(* Logix 5000 project; controller cal1615 1756-L62 rev 20.19; software revision 20.05; part 62 of 81 *)
(* tags used below, declared in another part *)
   FAULT : BOOL;   // Fault AFI
   HMI : BOOL;   // AFI HMI
   p01r09_pb_global_reset : BOOL;   // System Modes PB: Global Fault Reset
   p26_ao_dia_a : REAL;   // Upper Poly Letoff Analog Input Letoff A Diameter
   p26_ao_dia_b : REAL;   // Upper Poly Letoff Analog Input Letoff B Diameter
   p26_dint_to_hmi : DINT[16];   // Upper Poly Letoff Dint to HMI
   p26_ltf_a_sensor_input_max : REAL;
   p26_ltf_a_sensor_input_min : REAL;
   p26_ltf_a_sensor_output_max : REAL;
   p26_ltf_a_sensor_output_min : REAL;
   p26_ltf_b_sensor_input_max : REAL;
   p26_ltf_b_sensor_input_min : REAL;
   p26_ltf_b_sensor_output_max : REAL;
   p26_ltf_b_sensor_output_min : REAL;
   p26_ula_prs_input_max : REAL;
   p26_ula_prs_input_min : REAL;
   p26_ula_prs_output_max : REAL;
   p26_ula_prs_output_min : REAL;
   p26_ulb_prs_input_max : REAL;
   p26_ulb_prs_input_min : REAL;
   p26_ulb_prs_output_max : REAL;
   p26_ulb_prs_output_min : REAL;
   p26r01 : routine;   // Upper Poly Letoff
   p26r02 : routine;   // Upper Poly Letoff
   p26r02_fault_exists : BOOL;
   p26r02_timer_fault : TIMER[4];   // Upper Poly Letoff Misc Control Fault Delay
   p26r02_timer_warning : TIMER[4];   // Upper Poly Letoff Misc Control Warning Delay
   p26r02_unack_fault : BOOL;   // Upper Poly Letoff Misc Control Unacknowledged Fault Exists
   p26r02_unack_warning : BOOL;   // Upper Poly Letoff Misc Control Unacknowledged Warning Exists
   p26r02_warning_exists : BOOL;
   p26r03 : routine;   // Upper Poly Letoff Input
   p26r03_a_radius : REAL;
   p26r03_ai_dia_a_sensor : REAL;
   p26r03_ai_dia_b_sensor : REAL;
   p26r03_b_radius : REAL;
   p26r03_ltf_a_sensor_scp : SYS_SCP;   // Upper Poly Letoff Analog Input Diameter A Sensor Scaling
   p26r03_ltf_b_sensor_scp : SYS_SCP;   // Upper Poly Letoff Analog Input Letoff B Diameter Sensor Scaling
   p26r03_timer_fault : TIMER[4];   // Lower Poly Letoff Input Fault Delay
   p26r03_timer_warning : TIMER[4];   // Lower Poly Letoff Input Warning Delay
   p26r03_upper_A_tension_on : BOOL;
   p26r03_upper_B_tension_on : BOOL;
   p26r03_upper_poly_a_distance : REAL;
   p26r03_upper_poly_b_distance : REAL;
   p26r04 : routine;   // Upper Poly Letoff Output
   p26r04_timer_fault : TIMER[4];   // Lower Poly Letoff Output Fault Delay
   p26r04_timer_warning : TIMER[4];   // Lower Poly Letoff Output Warning Delay
   p26r04_ula_prs_scp : SYS_SCP;   // Upper Poly Lefoff Analog Output Letoff A Brake Pressure
   p26r04_ulb_prs_scp : SYS_SCP;   // Upper Poly Lefoff Analog Output Letoff B Brake Pressure
   p26r05 : routine;   // Upper Poly Letoff Dint to HMI
   p26r05_timer_fault : TIMER[4];   // Lower Poly Letoff Dint to HMI Fault Delay
   p26r06 : routine;   // Upper Poly Letoff Real to HMI
   p26r07 : routine;   // Upper Poly Letoff Alarms
   p26r08 : routine;   // Upper Poly Letoff Warnings
   p26r09 : routine;   // Upper Poly Letoff Modes
   p26r10 : routine;   // Upper Poly Letoff Tension
   p26r10_ula_selected_tension : REAL;   // Upper Poly Letoff Tension A Selected Tension
   p26r10_ulb_selected_tension : REAL;   // Upper Poly Letoff Tension B Selected Tension

PROGRAM P26_Upper_Poly_Letoff   (* main routine R01_Main *)

ROUTINE R01_Main   (* ladder *)
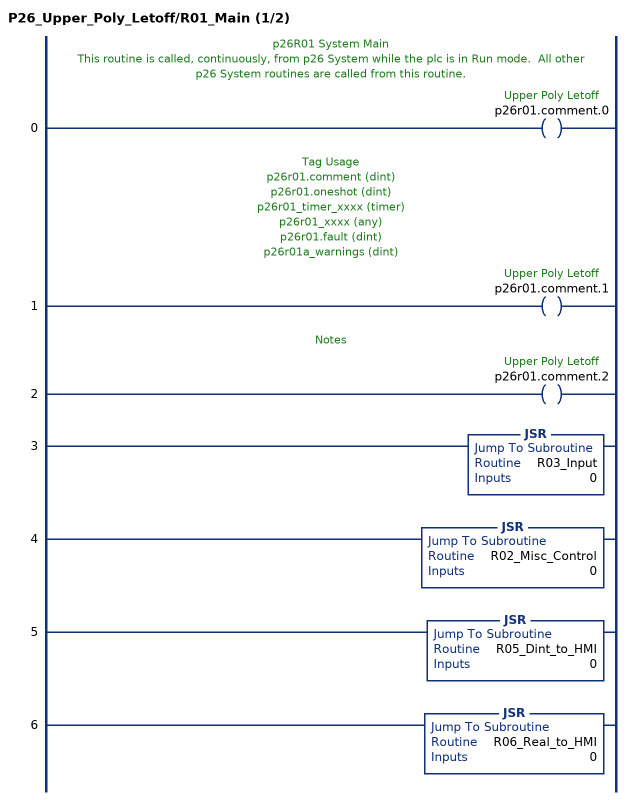
   // p26R01 System Main
   // This routine is called, continuously, from p26 System while the plc is in Run mode.  All other p26 System routines are called from this routine.
   0: OTE(p26r01.comment.0);
   // Tag Usage
   // p26r01.comment (dint)
   // p26r01.oneshot (dint)
   // p26r01_timer_xxxx (timer)
   // p26r01_xxxx (any)
   // p26r01.fault (dint)
   // p26r01a_warnings (dint)
   1: OTE(p26r01.comment.1);
   // Notes
   2: OTE(p26r01.comment.2);
   3: JSR(R03_Input,0);
   4: JSR(R02_Misc_Control,0);
   5: JSR(R05_Dint_to_HMI,0);
   6: JSR(R06_Real_to_HMI,0);
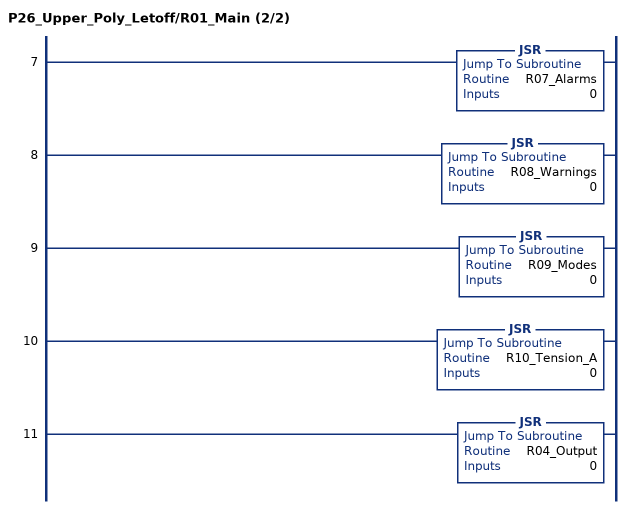
   7: JSR(R07_Alarms,0);
   8: JSR(R08_Warnings,0);
   9: JSR(R09_Modes,0);
   10: JSR(R10_Tension_A,0);
   11: JSR(R04_Output,0);
END_ROUTINE

ROUTINE R02_Misc_Control   (* ladder *)
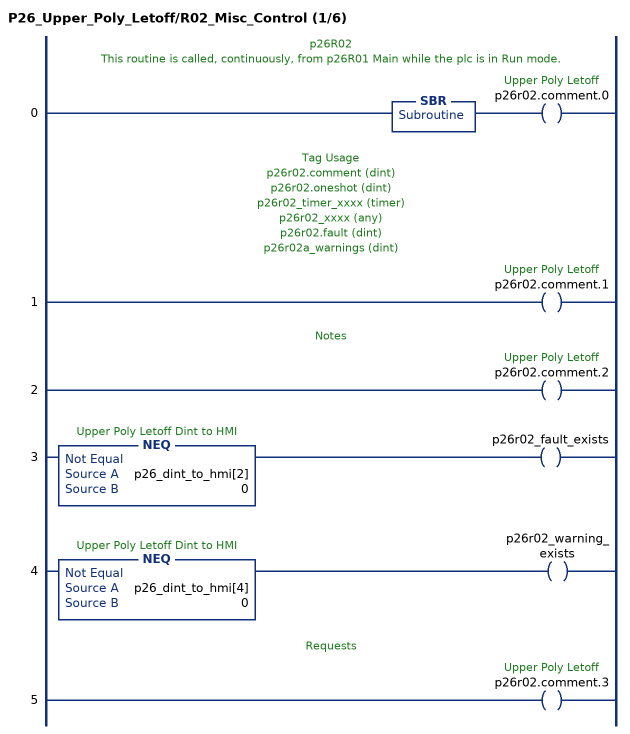
   // p26R02
   // This routine is called, continuously, from p26R01 Main while the plc is in Run mode.
   0: SBR()OTE(p26r02.comment.0);
   // Tag Usage
   // p26r02.comment (dint)
   // p26r02.oneshot (dint)
   // p26r02_timer_xxxx (timer)
   // p26r02_xxxx (any)
   // p26r02.fault (dint)
   // p26r02a_warnings (dint)
   1: OTE(p26r02.comment.1);
   // Notes
   2: OTE(p26r02.comment.2);
   3: NEQ(p26_dint_to_hmi[2],0)OTE(p26r02_fault_exists);
   4: NEQ(p26_dint_to_hmi[4],0)OTE(p26r02_warning_exists);
   // Requests
   5: OTE(p26r02.comment.3);
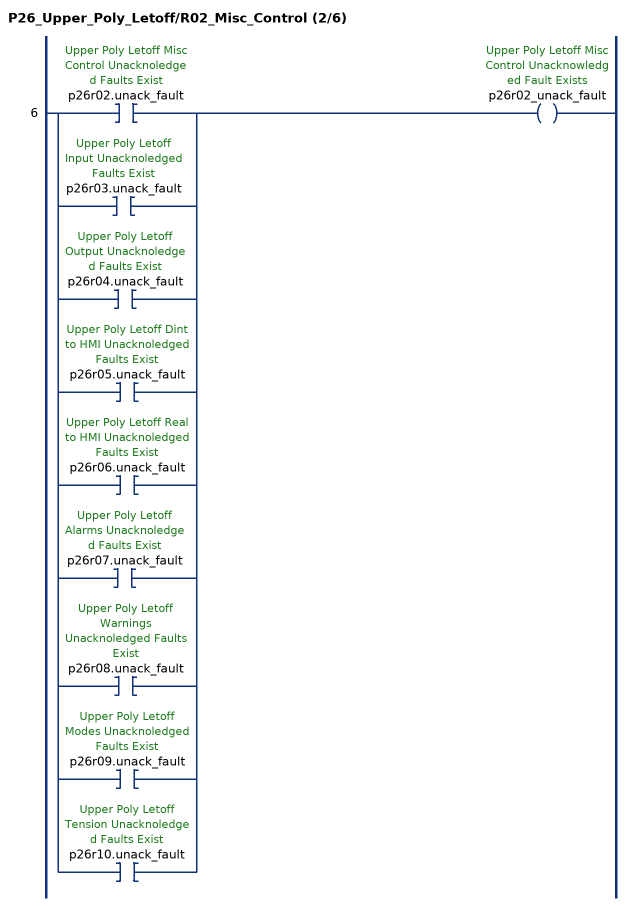
   6: [XIC(p26r02.unack_fault) ,XIC(p26r03.unack_fault) ,XIC(p26r04.unack_fault) ,XIC(p26r05.unack_fault) ,XIC(p26r06.unack_fault) ,XIC(p26r07.unack_fault) ,XIC(p26r08.unack_fault) ,XIC(p26r09.unack_fault) ,XIC(p26r10.unack_fault) ]OTE(p26r02_unack_fault);
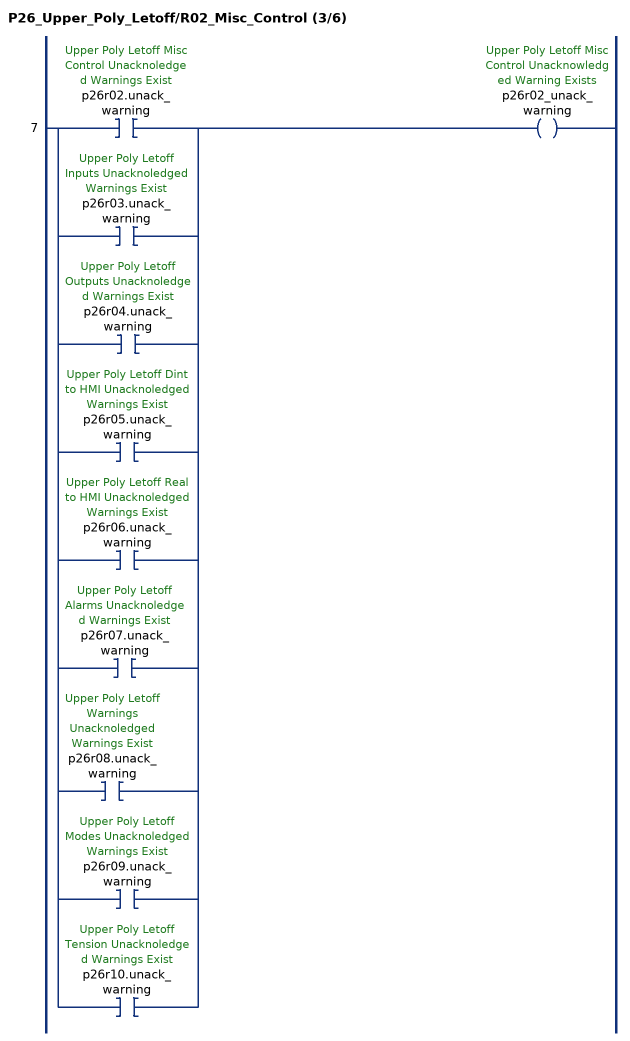
   7: [XIC(p26r02.unack_warning) ,XIC(p26r03.unack_warning) ,XIC(p26r04.unack_warning) ,XIC(p26r05.unack_warning) ,XIC(p26r06.unack_warning) ,XIC(p26r07.unack_warning) ,XIC(p26r08.unack_warning) ,XIC(p26r09.unack_warning) ,XIC(p26r10.unack_warning) ]OTE(p26r02_unack_warning);
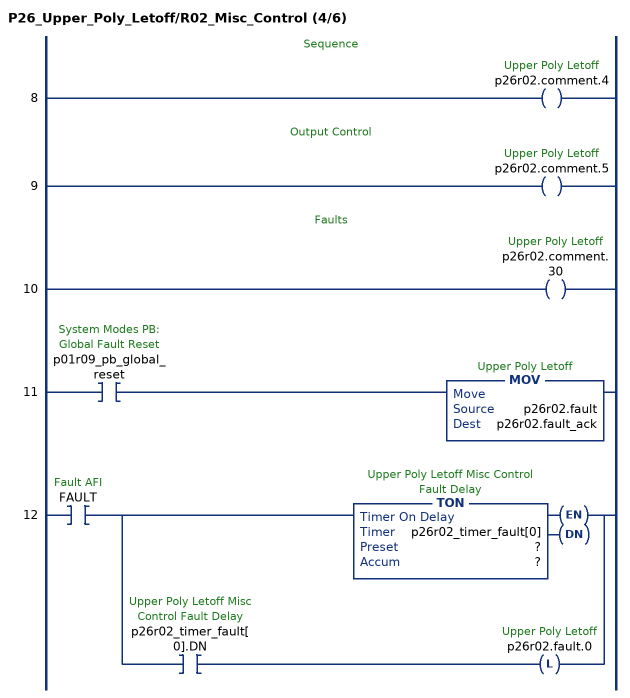
   // Sequence
   8: OTE(p26r02.comment.4);
   // Output Control
   9: OTE(p26r02.comment.5);
   // Faults
   10: OTE(p26r02.comment.30);
   11: XIC(p01r09_pb_global_reset)MOV(p26r02.fault,p26r02.fault_ack);
   12: XIC(FAULT)[TON(p26r02_timer_fault[0],?,?) ,XIC(p26r02_timer_fault[0].DN) OTL(p26r02.fault.0) ];
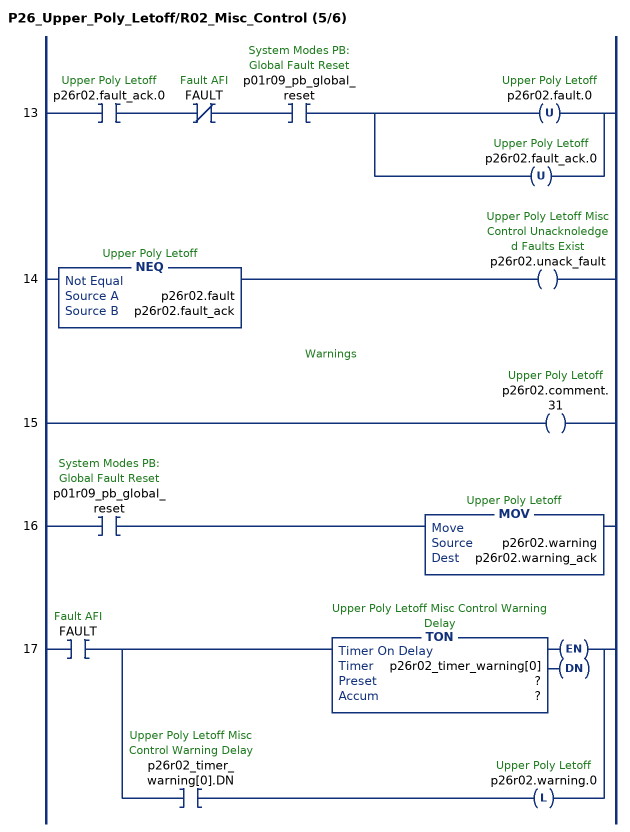
   13: XIC(p26r02.fault_ack.0)XIO(FAULT)XIC(p01r09_pb_global_reset)[OTU(p26r02.fault.0) ,OTU(p26r02.fault_ack.0) ];
   14: NEQ(p26r02.fault,p26r02.fault_ack)OTE(p26r02.unack_fault);
   // Warnings
   15: OTE(p26r02.comment.31);
   16: XIC(p01r09_pb_global_reset)MOV(p26r02.warning,p26r02.warning_ack);
   17: XIC(FAULT)[TON(p26r02_timer_warning[0],?,?) ,XIC(p26r02_timer_warning[0].DN) OTL(p26r02.warning.0) ];
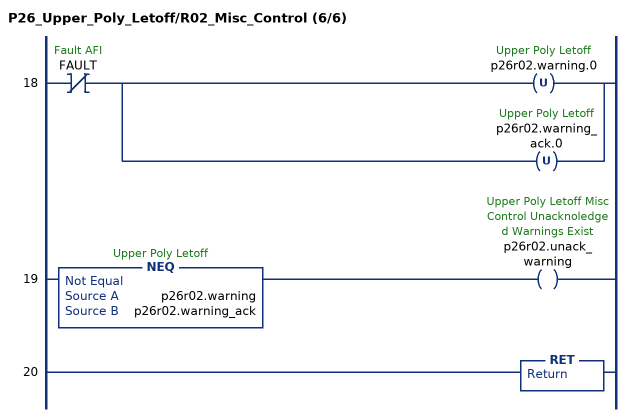
   18: XIO(FAULT)[OTU(p26r02.warning.0) ,OTU(p26r02.warning_ack.0) ];
   19: NEQ(p26r02.warning,p26r02.warning_ack)OTE(p26r02.unack_warning);
   20: RET();
END_ROUTINE

ROUTINE R03_Input   (* ladder *)
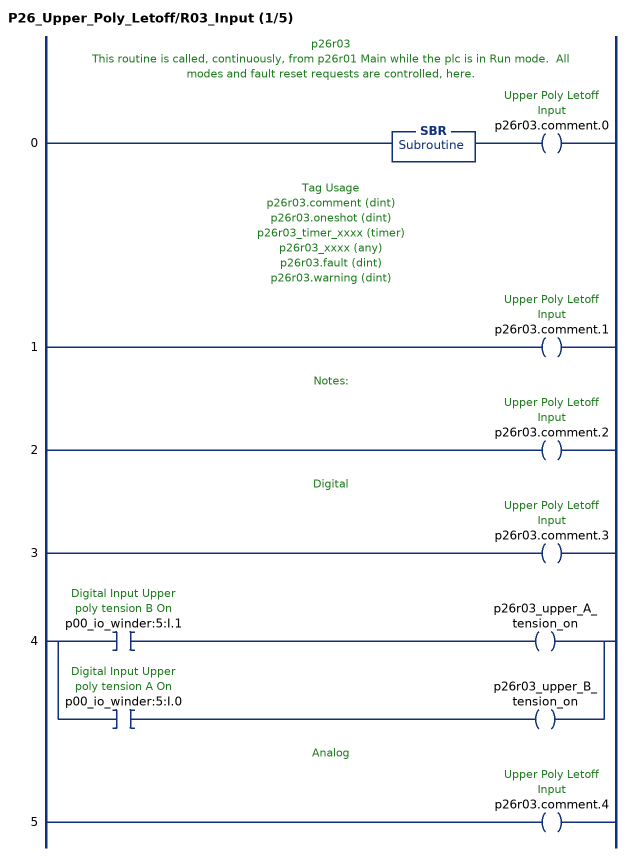
   // p26r03
   // This routine is called, continuously, from p26r01 Main while the plc is in Run mode.  All modes and fault reset requests are controlled, here.
   0: SBR()OTE(p26r03.comment.0);
   // Tag Usage
   // p26r03.comment (dint)
   // p26r03.oneshot (dint)
   // p26r03_timer_xxxx (timer)
   // p26r03_xxxx (any)
   // p26r03.fault (dint)
   // p26r03.warning (dint)
   1: OTE(p26r03.comment.1);
   // Notes:
   2: OTE(p26r03.comment.2);
   // Digital
   3: OTE(p26r03.comment.3);
   4: [XIC(p00_io_winder:5:I.1) OTE(p26r03_upper_A_tension_on) ,XIC(p00_io_winder:5:I.0) OTE(p26r03_upper_B_tension_on) ];
   // Analog
   5: OTE(p26r03.comment.4);
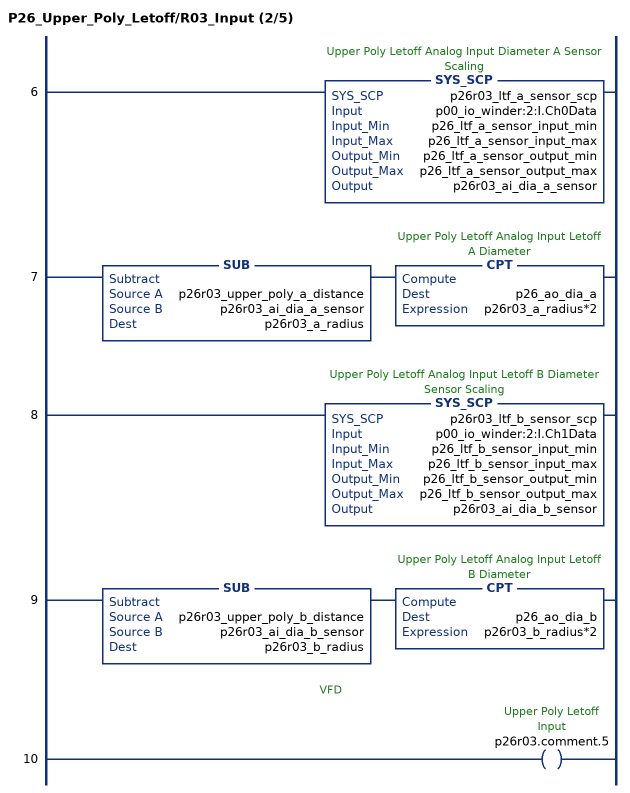
   6: SYS_SCP(p26r03_ltf_a_sensor_scp,p00_io_winder:2:I.Ch0Data,p26_ltf_a_sensor_input_min,p26_ltf_a_sensor_input_max,p26_ltf_a_sensor_output_min,p26_ltf_a_sensor_output_max,p26r03_ai_dia_a_sensor);
   7: SUB(p26r03_upper_poly_a_distance,p26r03_ai_dia_a_sensor,p26r03_a_radius)CPT(p26_ao_dia_a,p26r03_a_radius*2);
   8: SYS_SCP(p26r03_ltf_b_sensor_scp,p00_io_winder:2:I.Ch1Data,p26_ltf_b_sensor_input_min,p26_ltf_b_sensor_input_max,p26_ltf_b_sensor_output_min,p26_ltf_b_sensor_output_max,p26r03_ai_dia_b_sensor);
   9: SUB(p26r03_upper_poly_b_distance,p26r03_ai_dia_b_sensor,p26r03_b_radius)CPT(p26_ao_dia_b,p26r03_b_radius*2);
   // VFD
   10: OTE(p26r03.comment.5);
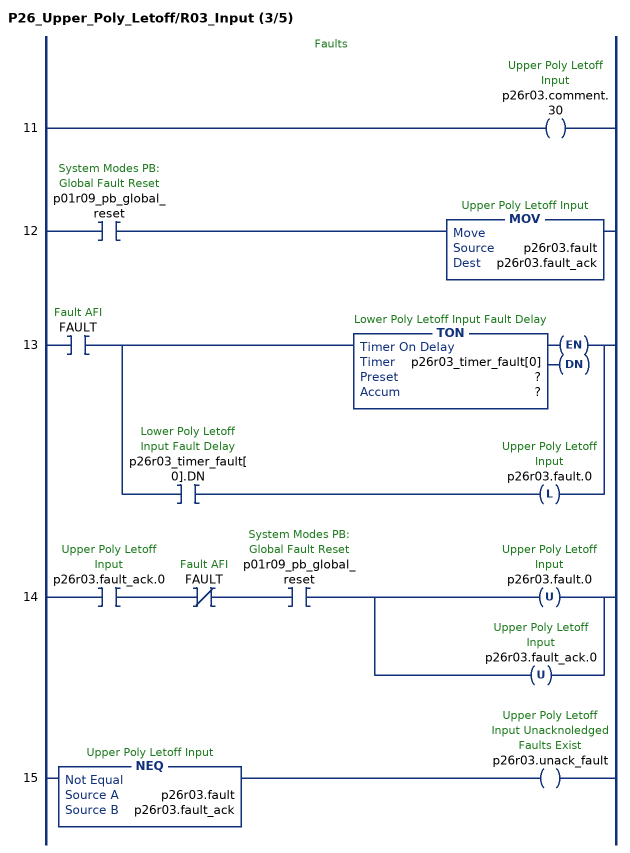
   // Faults
   11: OTE(p26r03.comment.30);
   12: XIC(p01r09_pb_global_reset)MOV(p26r03.fault,p26r03.fault_ack);
   13: XIC(FAULT)[TON(p26r03_timer_fault[0],?,?) ,XIC(p26r03_timer_fault[0].DN) OTL(p26r03.fault.0) ];
   14: XIC(p26r03.fault_ack.0)XIO(FAULT)XIC(p01r09_pb_global_reset)[OTU(p26r03.fault.0) ,OTU(p26r03.fault_ack.0) ];
   15: NEQ(p26r03.fault,p26r03.fault_ack)OTE(p26r03.unack_fault);
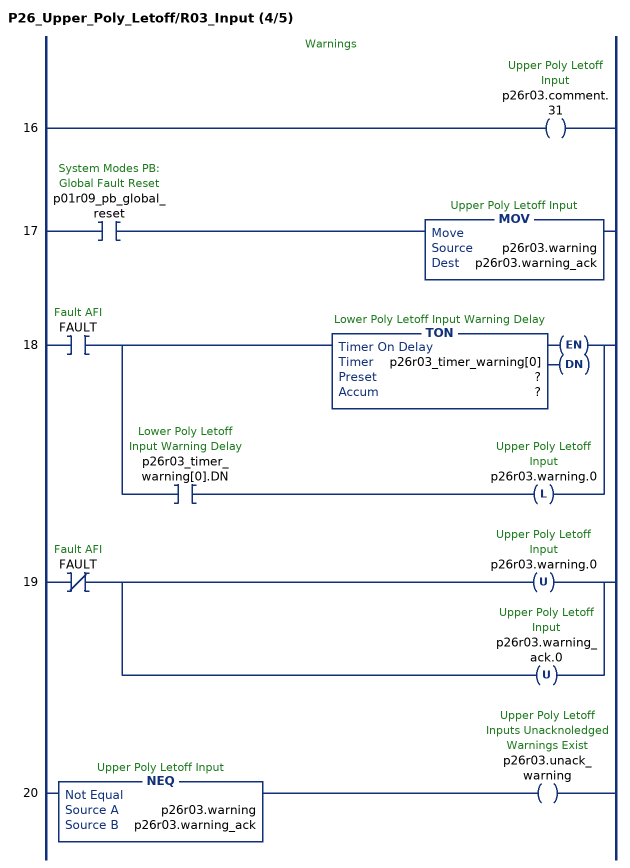
   // Warnings
   16: OTE(p26r03.comment.31);
   17: XIC(p01r09_pb_global_reset)MOV(p26r03.warning,p26r03.warning_ack);
   18: XIC(FAULT)[TON(p26r03_timer_warning[0],?,?) ,XIC(p26r03_timer_warning[0].DN) OTL(p26r03.warning.0) ];
   19: XIO(FAULT)[OTU(p26r03.warning.0) ,OTU(p26r03.warning_ack.0) ];
   20: NEQ(p26r03.warning,p26r03.warning_ack)OTE(p26r03.unack_warning);
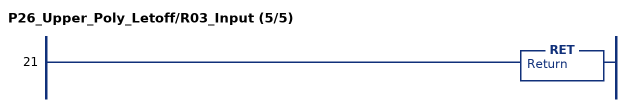
   21: RET();
END_ROUTINE

ROUTINE R04_Output   (* ladder *)
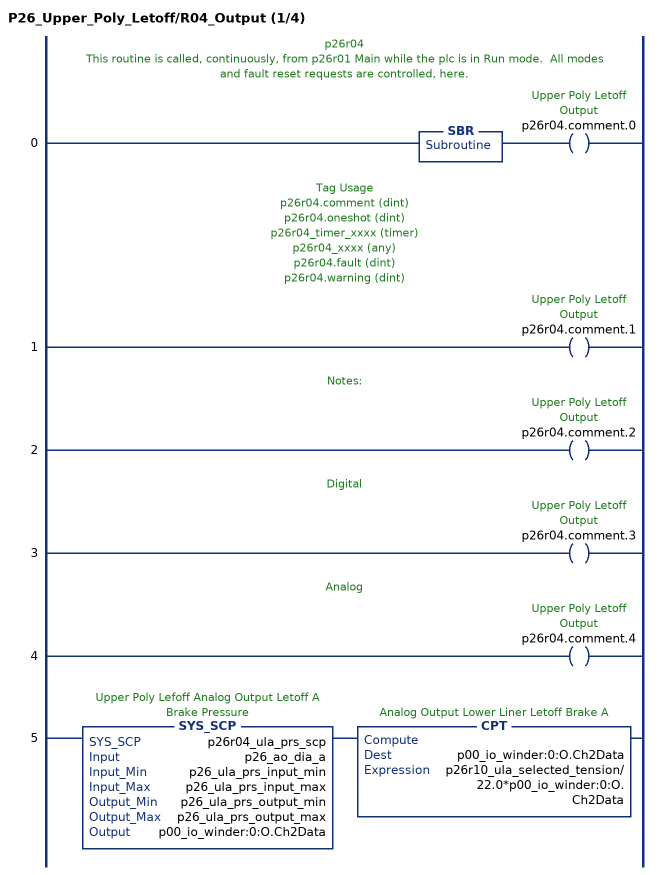
   // p26r04
   // This routine is called, continuously, from p26r01 Main while the plc is in Run mode.  All modes and fault reset requests are controlled, here.
   0: SBR()OTE(p26r04.comment.0);
   // Tag Usage
   // p26r04.comment (dint)
   // p26r04.oneshot (dint)
   // p26r04_timer_xxxx (timer)
   // p26r04_xxxx (any)
   // p26r04.fault (dint)
   // p26r04.warning (dint)
   1: OTE(p26r04.comment.1);
   // Notes:
   2: OTE(p26r04.comment.2);
   // Digital
   3: OTE(p26r04.comment.3);
   // Analog
   4: OTE(p26r04.comment.4);
   5: SYS_SCP(p26r04_ula_prs_scp,p26_ao_dia_a,p26_ula_prs_input_min,p26_ula_prs_input_max,p26_ula_prs_output_min,p26_ula_prs_output_max,p00_io_winder:0:O.Ch2Data)CPT(p00_io_winder:0:O.Ch2Data,p26r10_ula_selected_tension/22.0*p00_io_winder:0:O.Ch2Data);
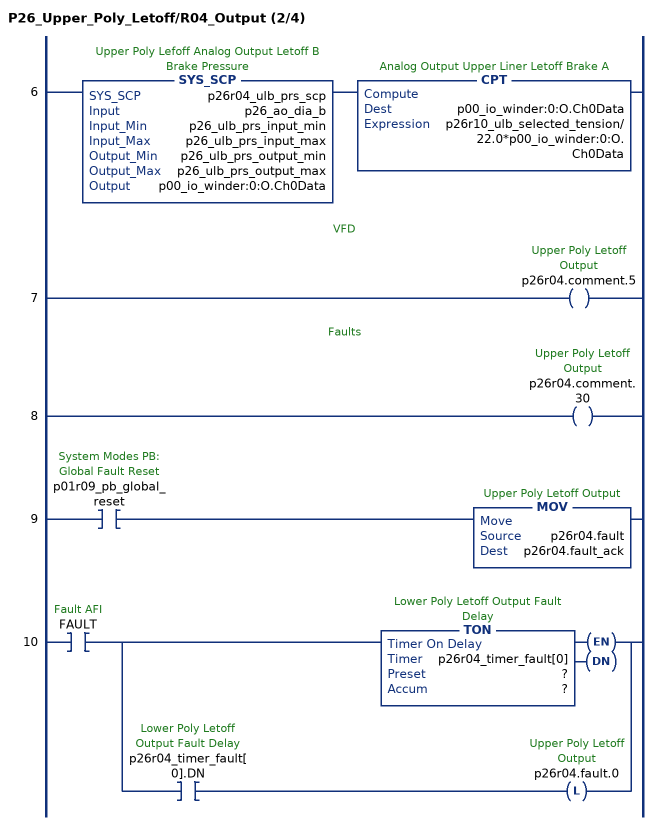
   6: SYS_SCP(p26r04_ulb_prs_scp,p26_ao_dia_b,p26_ulb_prs_input_min,p26_ulb_prs_input_max,p26_ulb_prs_output_min,p26_ulb_prs_output_max,p00_io_winder:0:O.Ch0Data)CPT(p00_io_winder:0:O.Ch0Data,p26r10_ulb_selected_tension/22.0*p00_io_winder:0:O.Ch0Data);
   // VFD
   7: OTE(p26r04.comment.5);
   // Faults
   8: OTE(p26r04.comment.30);
   9: XIC(p01r09_pb_global_reset)MOV(p26r04.fault,p26r04.fault_ack);
   10: XIC(FAULT)[TON(p26r04_timer_fault[0],?,?) ,XIC(p26r04_timer_fault[0].DN) OTL(p26r04.fault.0) ];
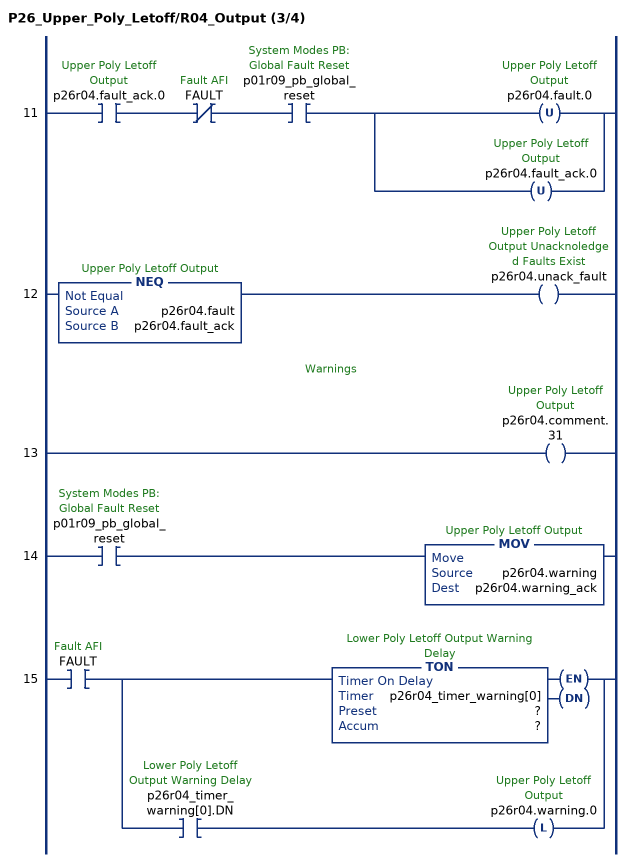
   11: XIC(p26r04.fault_ack.0)XIO(FAULT)XIC(p01r09_pb_global_reset)[OTU(p26r04.fault.0) ,OTU(p26r04.fault_ack.0) ];
   12: NEQ(p26r04.fault,p26r04.fault_ack)OTE(p26r04.unack_fault);
   // Warnings
   13: OTE(p26r04.comment.31);
   14: XIC(p01r09_pb_global_reset)MOV(p26r04.warning,p26r04.warning_ack);
   15: XIC(FAULT)[TON(p26r04_timer_warning[0],?,?) ,XIC(p26r04_timer_warning[0].DN) OTL(p26r04.warning.0) ];
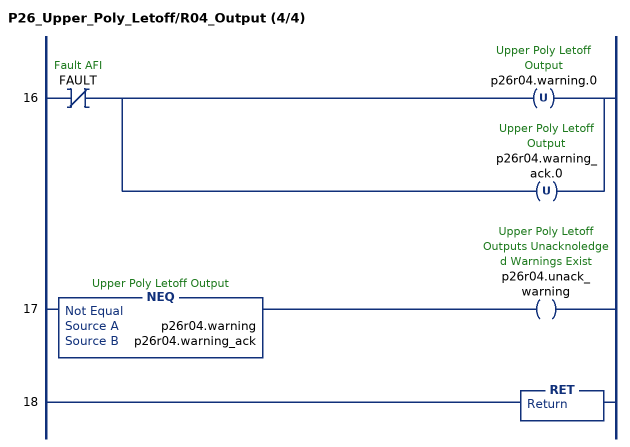
   16: XIO(FAULT)[OTU(p26r04.warning.0) ,OTU(p26r04.warning_ack.0) ];
   17: NEQ(p26r04.warning,p26r04.warning_ack)OTE(p26r04.unack_warning);
   18: RET();
END_ROUTINE

ROUTINE R05_Dint_to_HMI   (* ladder *)
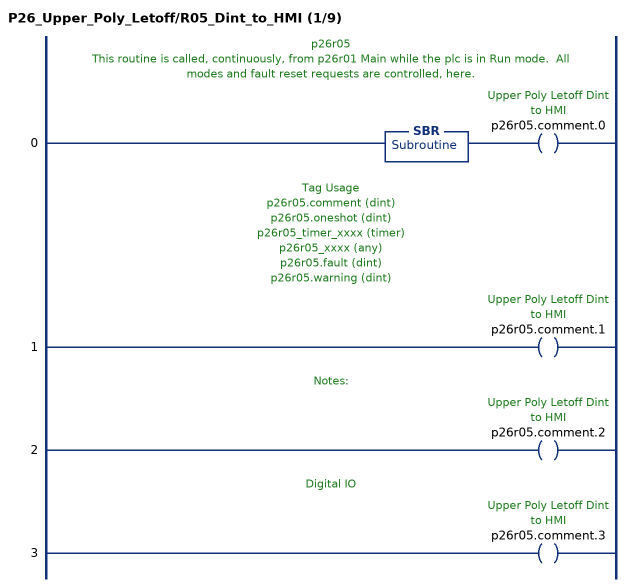
   // p26r05
   // This routine is called, continuously, from p26r01 Main while the plc is in Run mode.  All modes and fault reset requests are controlled, here.
   0: SBR()OTE(p26r05.comment.0);
   // Tag Usage
   // p26r05.comment (dint)
   // p26r05.oneshot (dint)
   // p26r05_timer_xxxx (timer)
   // p26r05_xxxx (any)
   // p26r05.fault (dint)
   // p26r05.warning (dint)
   1: OTE(p26r05.comment.1);
   // Notes:
   2: OTE(p26r05.comment.2);
   // Digital IO
   3: OTE(p26r05.comment.3);
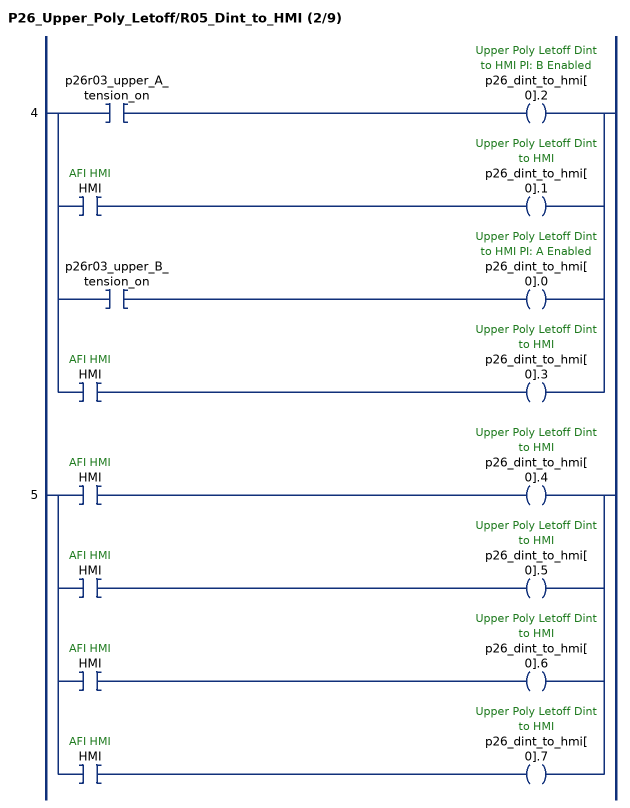
   4: [XIC(p26r03_upper_A_tension_on) OTE(p26_dint_to_hmi[0].2) ,XIC(HMI) OTE(p26_dint_to_hmi[0].1) ,XIC(p26r03_upper_B_tension_on) OTE(p26_dint_to_hmi[0].0) ,XIC(HMI) OTE(p26_dint_to_hmi[0].3) ];
   5: [XIC(HMI) OTE(p26_dint_to_hmi[0].4) ,XIC(HMI) OTE(p26_dint_to_hmi[0].5) ,XIC(HMI) OTE(p26_dint_to_hmi[0].6) ,XIC(HMI) OTE(p26_dint_to_hmi[0].7) ];
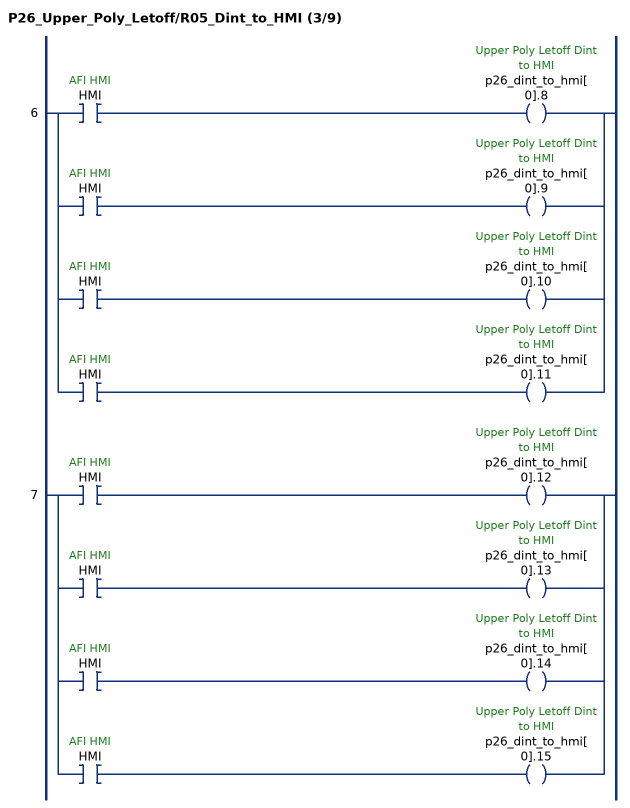
   6: [XIC(HMI) OTE(p26_dint_to_hmi[0].8) ,XIC(HMI) OTE(p26_dint_to_hmi[0].9) ,XIC(HMI) OTE(p26_dint_to_hmi[0].10) ,XIC(HMI) OTE(p26_dint_to_hmi[0].11) ];
   7: [XIC(HMI) OTE(p26_dint_to_hmi[0].12) ,XIC(HMI) OTE(p26_dint_to_hmi[0].13) ,XIC(HMI) OTE(p26_dint_to_hmi[0].14) ,XIC(HMI) OTE(p26_dint_to_hmi[0].15) ];
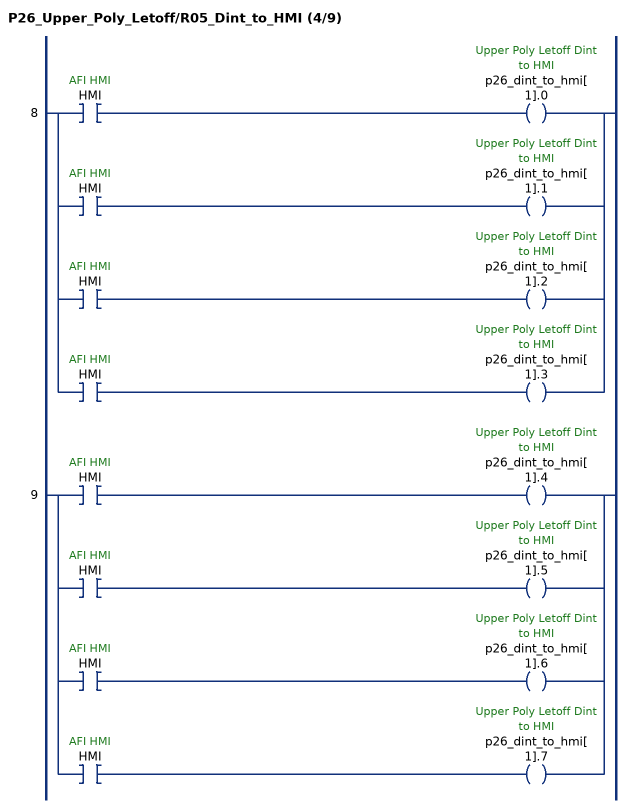
   8: [XIC(HMI) OTE(p26_dint_to_hmi[1].0) ,XIC(HMI) OTE(p26_dint_to_hmi[1].1) ,XIC(HMI) OTE(p26_dint_to_hmi[1].2) ,XIC(HMI) OTE(p26_dint_to_hmi[1].3) ];
   9: [XIC(HMI) OTE(p26_dint_to_hmi[1].4) ,XIC(HMI) OTE(p26_dint_to_hmi[1].5) ,XIC(HMI) OTE(p26_dint_to_hmi[1].6) ,XIC(HMI) OTE(p26_dint_to_hmi[1].7) ];
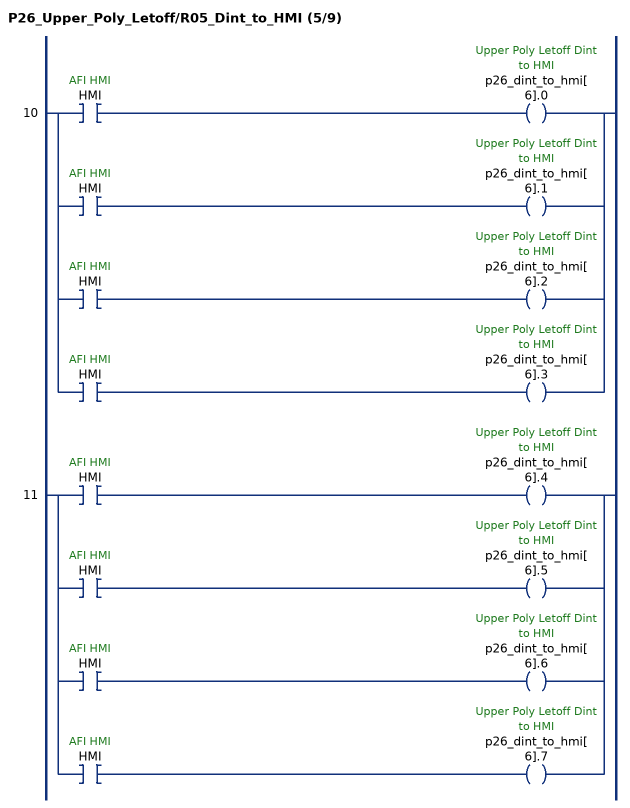
   10: [XIC(HMI) OTE(p26_dint_to_hmi[6].0) ,XIC(HMI) OTE(p26_dint_to_hmi[6].1) ,XIC(HMI) OTE(p26_dint_to_hmi[6].2) ,XIC(HMI) OTE(p26_dint_to_hmi[6].3) ];
   11: [XIC(HMI) OTE(p26_dint_to_hmi[6].4) ,XIC(HMI) OTE(p26_dint_to_hmi[6].5) ,XIC(HMI) OTE(p26_dint_to_hmi[6].6) ,XIC(HMI) OTE(p26_dint_to_hmi[6].7) ];
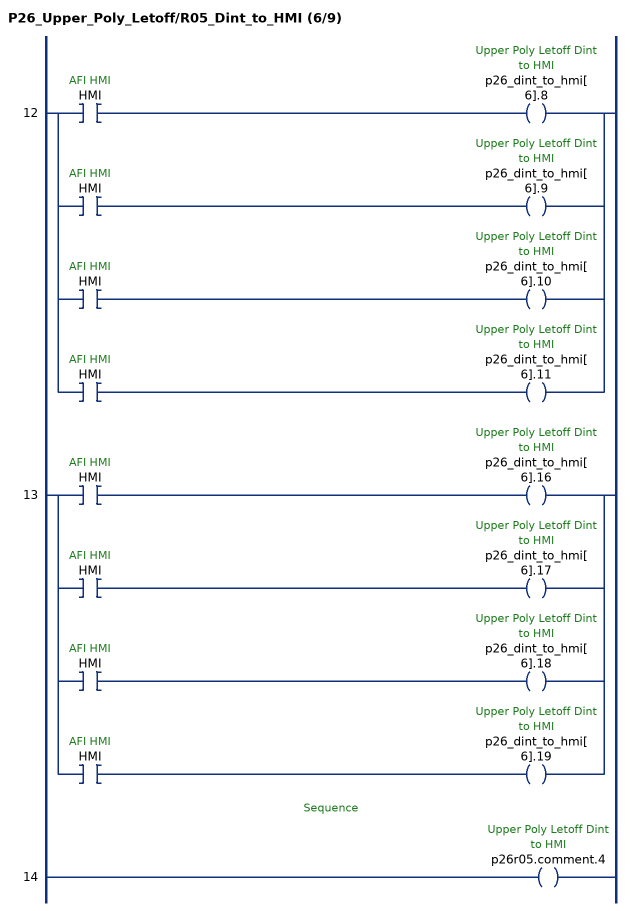
   12: [XIC(HMI) OTE(p26_dint_to_hmi[6].8) ,XIC(HMI) OTE(p26_dint_to_hmi[6].9) ,XIC(HMI) OTE(p26_dint_to_hmi[6].10) ,XIC(HMI) OTE(p26_dint_to_hmi[6].11) ];
   13: [XIC(HMI) OTE(p26_dint_to_hmi[6].16) ,XIC(HMI) OTE(p26_dint_to_hmi[6].17) ,XIC(HMI) OTE(p26_dint_to_hmi[6].18) ,XIC(HMI) OTE(p26_dint_to_hmi[6].19) ];
   // Sequence
   14: OTE(p26r05.comment.4);
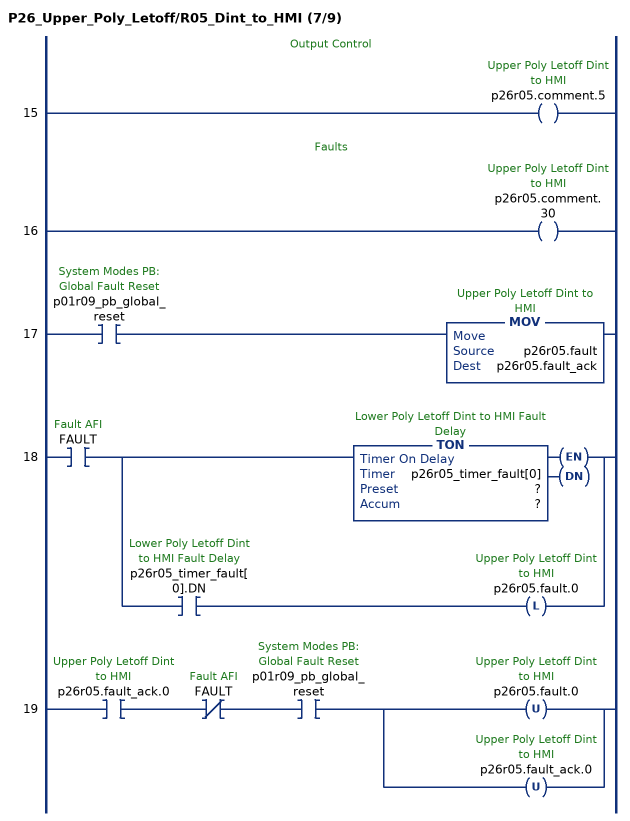
   // Output Control
   15: OTE(p26r05.comment.5);
   // Faults
   16: OTE(p26r05.comment.30);
   17: XIC(p01r09_pb_global_reset)MOV(p26r05.fault,p26r05.fault_ack);
   18: XIC(FAULT)[TON(p26r05_timer_fault[0],?,?) ,XIC(p26r05_timer_fault[0].DN) OTL(p26r05.fault.0) ];
   19: XIC(p26r05.fault_ack.0)XIO(FAULT)XIC(p01r09_pb_global_reset)[OTU(p26r05.fault.0) ,OTU(p26r05.fault_ack.0) ];
